FUNCTION_BLOCK Init_Condition (* Composite Function Block Type *)
  (* Standard: 61499-2; Description: InitEvent nya disambungin ke cold/warm aja ya SubsequentEvent nya disambungin ke event yg seharusnya *)
  (* Version 0.0, 2018-07-28, 4DIAC-IDE, 4DIAC-Consortium *)
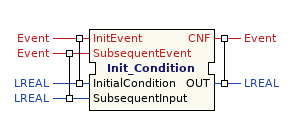
  EVENT_INPUT
    InitEvent WITH InitialCondition;
    SubsequentEvent WITH SubsequentInput;
  END_EVENT
  EVENT_OUTPUT
    CNF WITH OUT; (* Execution Confirmation *)
  END_EVENT
  VAR_INPUT
    InitialCondition : LREAL;
    SubsequentInput : LREAL;
  END_VAR
  VAR_OUTPUT
    OUT : LREAL;
  END_VAR
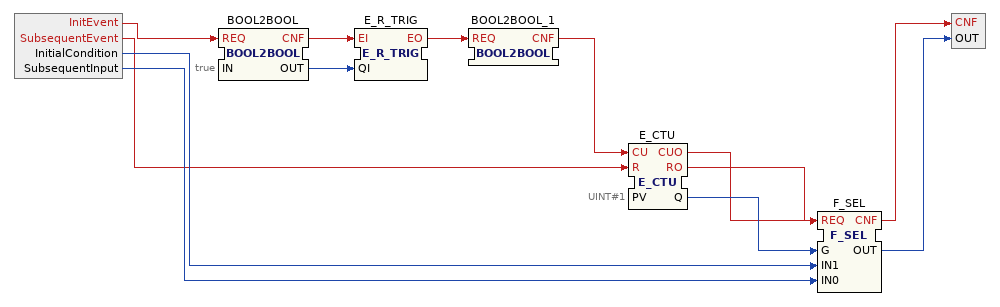
  FBS
    E_CTU : E_CTU(PV := UINT#1);
    BOOL2BOOL : BOOL2BOOL(IN := true);
    BOOL2BOOL_1 : BOOL2BOOL;
    E_R_TRIG : E_R_TRIG;
    F_SEL : F_SEL;
  END_FBS
  EVENT_CONNECTIONS
    InitEvent TO BOOL2BOOL.REQ;
    BOOL2BOOL.CNF TO E_R_TRIG.EI;
    E_R_TRIG.EO TO BOOL2BOOL_1.REQ;
    BOOL2BOOL_1.CNF TO E_CTU.CU;
    E_CTU.CUO TO F_SEL.REQ;
    E_CTU.RO TO F_SEL.REQ;
    SubsequentEvent TO E_CTU.R;
    F_SEL.CNF TO CNF;
  END_CONNECTIONS
  DATA_CONNECTIONS
    E_CTU.Q TO F_SEL.G;
    InitialCondition TO F_SEL.IN1;
    SubsequentInput TO F_SEL.IN0;
    F_SEL.OUT TO OUT;
    BOOL2BOOL.OUT TO E_R_TRIG.QI;
  END_CONNECTIONS
END_FUNCTION_BLOCK
